{attribute 'qualified_only'}
{attribute 'strict'}
{attribute 'to_string'}
TYPE E_3002_2_Inactive_Active : (
		Inactive := 0,
		Active	 := 1
	) UINT;
END_TYPE

(* stored: Version 1.1.0.1
   DUT E_3002_2_Inactive_Active: Id {7d1b6ada-9be7-45b0-9609-f0cb032d6919} *)
